TYPE typeStationEnables :
STRUCT
	McEnabled: BOOL;
	S1Enabled: BOOL;
	S2Enabled: BOOL;
	S3Enabled: BOOL;
	S4Enabled: BOOL;
	S5Enabled: BOOL;
	S6Enabled: BOOL;
END_STRUCT
END_TYPE

(* stored: Version 1.1.0.1, ProductVersion 3.1.4024.12
   DUT typeStationEnables: Id {687be2b5-dddf-440b-a143-f8846c13a1c9} *)
